FUNCTION_BLOCK FB_GovernorSerialCom
VAR
	sName			:		STRING;
	bInitialized	:		BOOL;
	iScantime		:		UINT;
	iTimeout		:		UINT;
	
	bBusy			: 		BOOL;
	bError			:		BOOL;
	
	iStepInit		:		INT;
	iStepGeneral	: 		INT;
	iStepRunning	:		INT;
	bFirstCycle		:		BOOL := TRUE;
	
	bRun			:		BOOL;
	bStop			: 		BOOL;
	
	fbSendData		: 		SendData;
	fbReadData		:		ReceiveData;
	fbPcComCtrl		:		SerialLineControl;
	pData			:		POINTER TO BYTE;
	iLength			:		UDINT;
	txBuffer		:		ComBuffer;
	rxBuffer		:		ComBuffer;
	stIn_PcCom AT %I*	: PcComInData;	
	stOut_PcCom AT %Q*	: PcComOutData;	
		
	sStationNo		:		ARRAY [0..1] OF BYTE := [16#30, 16#31];
	sPCNo			:		ARRAY [0..1] OF BYTE := [16#FF, 16#FF];
	sDeviceAdr		:		ARRAY [0..4] OF BYTE := [16#44, 16#30, 16#31, 16#36, 16#30];
	sNumberDevice	:		ARRAY [0..1] OF BYTE := [16#30, 16#37]; 
	
	stBatchReadFrame	:	U_GovernorSerialBatchRead;
	stAckFrame			:	U_GovernorSerialAck;
	stBatchResponseFrame:	U_GovernorSerialBatchResponse;
	
	bDelayState		:		BOOL;
	tonScanTime		:		TON;
	iLoop			:		INT;
	trSend			:		R_TRIG;
	
	a : WORD;
END_VAR
VAR CONSTANT
	iReadPrefix 	:	BYTE := 16#02;
	sCommandBatchRead	:	ARRAY [0..1] OF BYTE := [16#42, 16#52];
END_VAR

 IF bFirstCycle THEN
	bFirstCycle := FALSE;
	
	stBatchReadFrame.stFrame.iPrefix 	:= 16#05;
	stBatchReadFrame.stFrame.iStationNo := sStationNo;
	stBatchReadFrame.stFrame.iPCNo		:= sPCNo;
	stBatchReadFrame.stFrame.iCmdBatchRead := sCommandBatchRead;
	stBatchReadFrame.stFrame.iMsgWaitTime := 16#30;
	stBatchReadFrame.stFrame.iDeviceAdr	:= sDeviceAdr;
	stBatchReadFrame.stFrame.iNumberDevice := sNumberDevice;
	stBatchReadFrame.stFrame.iCheckSum[0] := WORD_TO_BYTE(SHR(F_CheckSum16(ADR(stBatchReadFrame) + 1, 14, 0), 4) AND 16#000F);
	stBatchReadFrame.stFrame.iCheckSum[1] := WORD_TO_BYTE(F_CheckSum16(ADR(stBatchReadFrame) + 1, 14, 0) AND 16#000F);
	
	stAckFrame.stFrame.iPrefix 		:= 16#06;
	stAckFrame.stFrame.iStationNo 	:= sStationNo;
	stAckFrame.stFrame.iPCNo 		:= sPCNo;
END_IF
		
StateMachine();

bInitialized := iStepGeneral >= 20;
bBusy := fbSendData.Busy AND fbReadData.busy AND iStepGeneral = 30;

bError S= (fbSendData.Error <> ComError_t.COMERROR_NOERROR OR fbReadData.Error <> ComError_t.COMERROR_NOERROR OR fbPcComCtrl.Error) AND (iStepGeneral = 30) AND (iStepRunning = 60);
bError R= (NOT (fbSendData.Error <> ComError_t.COMERROR_NOERROR) AND NOT (fbReadData.Error <> ComError_t.COMERROR_NOERROR) AND NOT fbPcComCtrl.Error) AND (iStepGeneral = 30) AND (iStepRunning = 60);

IF trSend.Q THEN
	fbSendData(pSendData := ADR(stBatchReadFrame), Length := SIZEOF(stBatchReadFrame), TXbuffer := txBuffer);
END_IF

fbReadData(
	pPrefix:= ADR(iReadPrefix),
	LenPrefix := 1,
	pReceiveData := ADR(stBatchResponseFrame),
	SizeReceiveData := SIZEOF(stBatchResponseFrame),
	Timeout:= T#1S,
	RXbuffer:= RxBuffer );
	
fbPcComCtrl(
	Mode:= SERIALLINEMODE_PC_COM_PORT, 
	pComIn:= ADR(stIn_PcCom), 
	pComOut:= ADR(stOut_PcCom), 
	SizeComIn:= SIZEOF(stIn_PcCom), 
	TxBuffer:= txBuffer, 
	RxBuffer:= rxBuffer );
	
tonScanTime(IN := iStepRunning >= 10 AND iStepRunning <= 100 AND iStepGeneral = 30, PT := INT_TO_TIME(iScantime));
trSend(CLK := iStepRunning >= 20 AND iStepRunning <= 30);

bRun := FALSE;
bStop := FALSE;

//	// error	
//		fbAxisError.Description := FUN_MergeStrings5(sMotorName, ' axis error number: ', UDINT_TO_STRING(iErrorID), '', '');
//		fbAxisError.Set(bError);

METHOD Abort : BOOL
END_METHOD

PROPERTY AnyError : BOOL
GET
AnyError 	:= bError;
END_GET
END_PROPERTY

PROPERTY Busy : BOOL
GET
Busy := bBusy;
END_GET
END_PROPERTY

PROPERTY DataBladeOpening : REAL
GET
DataBladeOpening := WORD_TO_REAL(stBatchResponseFrame.stFrame.iDataBladeOpening)/4096*100;
END_GET
END_PROPERTY

PROPERTY DataFrequency : REAL
GET
DataFrequency := WORD_TO_REAL(stBatchResponseFrame.stFrame.iDataFrequency)/32767*100;
END_GET
END_PROPERTY

PROPERTY DataGateOpening : REAL
GET
DataGateOpening := WORD_TO_REAL(stBatchResponseFrame.stFrame.iDataGateOpening)/4096*100;
END_GET
END_PROPERTY

PROPERTY DataGateOpenSet : REAL
GET
DataGateOpenSet := WORD_TO_REAL(stBatchResponseFrame.stFrame.iDataGateOpenSet)/32767*100;
END_GET
END_PROPERTY

PROPERTY DataState : WORD
GET
DataState := stBatchResponseFrame.stFrame.iDataState;
END_GET
END_PROPERTY

METHOD FirstCycle : BOOL
VAR_INPUT
//	ipAlarmController	: I_AlarmController;
//	ipHMIController	: I_HMIController;
END_VAR
END_METHOD

METHOD Init : BOOL
IF iStepGeneral = 0 THEN
	iStepGeneral := 10;
END_IF

//Method output
	Init := (iStepGeneral >= 20);
END_METHOD

PROPERTY Initialized : BOOL
GET
Initialized := bInitialized;
END_GET
END_PROPERTY

PROPERTY Name : STRING
GET
Name := sName;
END_GET
SET
sName := Name;
END_SET
END_PROPERTY

METHOD Reset : BOOL
bError := FALSE;
bError := FALSE;
iStepInit		:= 0;
iStepGeneral	:= 0;
iStepRunning	:= 0;


Reset := TRUE;
END_METHOD

METHOD Run : BOOL
IF (iStepGeneral = 20) THEN
	iStepGeneral := 30;
END_IF

bRun := TRUE;
Run := (iStepGeneral >= 30) AND (iStepGeneral < 200);
END_METHOD

PROPERTY ScanTime : UINT
GET
ScanTime := iScantime;
END_GET
SET
iScantime := ScanTime;
END_SET
END_PROPERTY

METHOD StateInit : BOOL (*Unit is performing initialization*)
IF NOT bError THEN
	iStepGeneral := 20;
END_IF
END_METHOD

METHOD StateMachine : BOOL (*State machine of unit*)
//State machine						   
	CASE iStepGeneral OF
		0:  //Uninitialized
			StateUninitialized();
	
		10: //Initializing
			StateInit();
	
		20: //Ready
			StateReady();
		
		30: //Running
			StateRunning();
						
		200: //stop
			StateStopping();
			
		210: //stop done
			StateStoppingDone();
	END_CASE
END_METHOD

METHOD StateReady : BOOL (* Unit is initialized*)
END_METHOD

METHOD StateRunning : BOOL (* Unit is uninitialized*)
VAR 
END_VAR
CASE iStepRunning OF
	0: // Trigger
		IF TRUE THEN
			iStepRunning := 10;
		END_IF

	10: // Request Send
		IF NOT fbSendData.Busy THEN
			iStepRunning := 20;
		END_IF
		
	20: // Confirm Send Request
		IF fbSendData.Busy THEN
			iStepRunning := 30;
		END_IF
		
	30: // Wait Send done
		IF NOT fbSendData.Busy THEN
			iStepRunning := 40;
		END_IF
		
	40: // Wait Receive event
		IF fbReadData.busy THEN
			iStepRunning := 50;
		END_IF
	
	50: // Wait Receive done
		IF NOT fbReadData.DataReceived THEN
			iStepRunning := 60;
		END_IF
		
	60: // Request Ack
		IF NOT fbSendData.Busy THEN
			iStepRunning := 70;
		END_IF
		
	70: // Confirm Ack
		IF fbSendData.Busy THEN
			iStepRunning := 80;
		END_IF
		
	80: // Wait Ack done
		IF NOT fbSendData.Busy THEN
			iStepRunning := 90;
		END_IF
		
	90: // Convert Data
		IF TRUE THEN
			iStepRunning := 100;
		END_IF
	
	100: // Return, done
		IF tonScanTime.Q THEN
			iStepRunning := 0;
		END_IF
	
END_CASE
END_METHOD

METHOD StateStopping : BOOL (* Unit is uninitialized*)
iStepGeneral	:= 210;
iStepRunning	:= 0;
END_METHOD

METHOD StateStoppingDone : BOOL (* Unit is uninitialized*)
IF NOT bStop THEN
	iStepGeneral := 20;
END_IF
END_METHOD

METHOD StateUninitialized : BOOL (* Unit is uninitialized*)
END_METHOD

METHOD Stop : BOOL
IF iStepGeneral >= 30 AND iStepGeneral < 200 THEN
	iStepGeneral := 200;
END_IF
bStop := TRUE;

Stop := (iStepGeneral = 210);
END_METHOD

PROPERTY Timeout : UINT
GET
Timeout := iTimeout;
END_GET
SET
iTimeout := Timeout;
END_SET
END_PROPERTY

END_FUNCTION_BLOCK

(* stored: Version 1.1.0.1, ProductVersion 3.1.4024.12
   POU FB_GovernorSerialCom: Id {52a5f590-92ea-4c20-8cb3-84d054e3fd22}, SpecialFunc None
   Folder Methods: Id {84fc7178-4e1b-4d9a-bc3b-4a5afe5bf133}
   Folder Properties: Id {b0cde6b9-b1bc-4db2-b0f5-1f26e810666c}
   Folder Data: Id {9d42a754-4192-44df-a725-bb30cb51e009}
   Folder StateMachine: Id {9b1a1034-2123-4a43-8ff9-221c46ed01fb}
   Method Abort: Id {ac029164-0da0-4543-9d43-0f26c5ad1003}
   Property AnyError: Id {4e6f9141-7e35-4a9f-8921-ee4f84dd0827}
   Get Get: Id {9ad3e1dd-a044-4326-81d8-9ff5b0038567}
   Property Busy: Id {f071631c-b89d-4a14-9b33-2744b501ade2}
   Get Get: Id {59ac161d-3510-4e9e-a694-cf1af4e330c3}
   Property DataBladeOpening: Id {67d0e371-25b0-4037-885b-7c165fddd147}
   Get Get: Id {02fd01de-dd4c-415a-aa64-62f219258194}
   Property DataFrequency: Id {5032ac4e-edc3-4a60-9c97-907ddd57d20e}
   Get Get: Id {150f917b-c83b-4146-a976-b6c74dc69d4c}
   Property DataGateOpening: Id {b72f232f-7bbf-4da0-a6ec-7f113ecdef66}
   Get Get: Id {077137ec-abc1-462c-a724-4e45db4096b3}
   Property DataGateOpenSet: Id {004b4d17-3045-41ac-bb85-e5dd1883263b}
   Get Get: Id {713ff82e-751a-4110-b51d-54f5c87110b7}
   Property DataState: Id {911ff35f-f606-42c7-be5f-4da6a512535d}
   Get Get: Id {2f847ecb-d988-4738-8844-226dd2816980}
   Method FirstCycle: Id {fb0033be-add6-483f-b39a-5e7a9cf9e853}
   Method Init: Id {26ebf153-e11e-47d6-aba9-17bcec119ceb}
   Property Initialized: Id {ecf18dd1-c2d9-4232-b1d8-a740c89b4693}
   Get Get: Id {2fe62b97-a097-4539-b4e4-d92bc4daada9}
   Property Name: Id {5e745e47-3a98-4a44-91d9-3b550cceacfb}
   Get Get: Id {0c4799de-2d4e-4105-b9e3-115d293d9a57}
   Set Set: Id {ee588da0-b295-4569-8946-3626e9442c9c}
   Method Reset: Id {9c86d807-994f-4463-8118-361821ba586e}
   Method Run: Id {c79f7041-73ae-430c-9dcf-78d249b0e3bf}
   Property ScanTime: Id {bd649d1c-bc52-4a29-ab0a-2b0c80efb6c4}
   Get Get: Id {01f11b07-25ce-4fc5-abc3-96a15629b4a8}
   Set Set: Id {1cd8a04e-d694-403e-8e66-c84414ea117c}
   Method StateInit: Id {2fc89dfb-53ac-489a-9393-a850a4ce0ad1}
   Method StateMachine: Id {c054500d-4632-46b0-95ab-2b1b14e2f7f2}
   Method StateReady: Id {97354b86-a8aa-4b1d-98d3-b12c9b305662}
   Method StateRunning: Id {8064ce6a-a2b6-4712-8f1b-ecf606b53326}
   Method StateStopping: Id {88cc0c69-2e36-4116-9317-cc3aa8ea1889}
   Method StateStoppingDone: Id {99505961-561c-466d-ad55-50e67aede28a}
   Method StateUninitialized: Id {b2bc5e98-e8d0-4aad-a3a9-b266a482fce2}
   Method Stop: Id {da0dfe7c-bfeb-446c-a827-2a61440e887c}
   Property Timeout: Id {0307c532-c249-4641-8d41-8c13eefdb92b}
   Get Get: Id {7ab159e1-75c3-4531-b797-12b78d30ff8f}
   Set Set: Id {ebd85a5b-ae9b-4ebc-bd89-5cbd88ab23f0} *)
